// TIA Portal V16 export
// export: Created 2020-03-15T18:15:52.6815683Z, ExportSetting WithDefaults, WithReadOnly, DisplayName Totally Integrated Automation Portal, DisplayVersion V16, DisplayName TIA Portal Version Control Interface, DisplayVersion V16, DisplayName TIA Portal Openness, DisplayVersion V16, DisplayName STEP 7 Professional, DisplayVersion V16, DisplayName STEP 7 Safety, DisplayVersion V16, DisplayName WinCC Advanced, DisplayVersion V16
TYPE "Step"
// stored: CreationDate 2020-03-15T11:44:40.2322714Z, InterfaceModifiedDate 2020-03-15T17:59:49.5298338Z, IsConsistent true, IsFailsafeCompliant false, IsKnowHowProtected false, LibraryConformanceStatus Das Objekt ist bibliothekskonform., ModifiedDate 2020-03-15T18:05:07.0457628Z
   STRUCT
      Next : Int;   // next step no.
      Abort : Int;   // abort step no.
      Option1 : Int;   // optional step 1
      Option2 : Int;   // optional step 2
      MonitorTime : Int;   // max. time step
      "Name" : WString[20];   // name of the step
      WaitingTime : DInt;   // wainting time
   END_STRUCT;
END_TYPE
